# EPICS substitutions: iocvcs/iocvcsApp/Db/userHost.substitutions
# Example substitutions file

file "db/dbExample1.db" {
    { user = "yannHost" }
}

file db/dbExample2.db {
    pattern { user, no, scan }
        { "yannHost", 1, "1 second" }
        { "yannHost", 2, "2 second" }
        { "yannHost", 3, "5 second" }
}
